// Mitsubishi GX Works2 project: ConcentricityP202112270800   PLC: Q03UDV

PROGRAM 1_AUTO
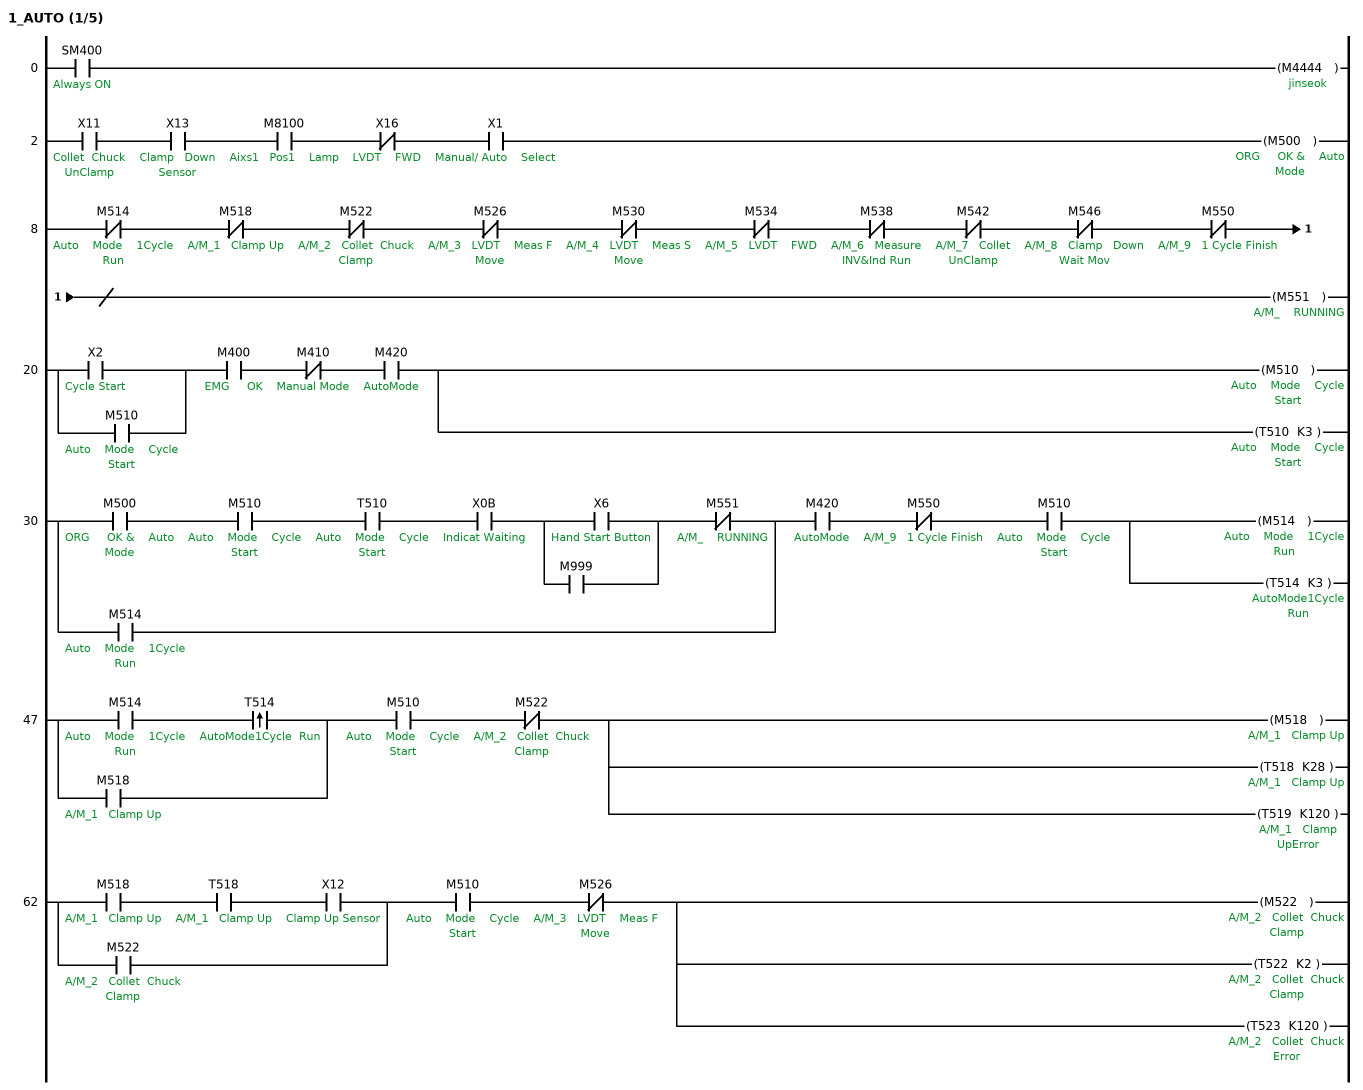
0     LD      SM400  ; Always ON
      OUT     M4444  ; jinseok
2     LD      X11  ; Collet  Chuck   UnClamp
      AND     X13  ; Clamp   Down    Sensor
      AND     M8100  ; Aixs1   Pos1    Lamp
      ANI     X16  ; LVDT    FWD
      AND     X1  ; Manual/ Auto    Select
      OUT     M500  ; ORG     OK &    Auto    Mode
8     LDI     M514  ; Auto    Mode    1Cycle  Run
      ANI     M518  ; A/M_1   Clamp Up
      ANI     M522  ; A/M_2   Collet  Chuck   Clamp
      ANI     M526  ; A/M_3   LVDT    Meas F  Move
      ANI     M530  ; A/M_4   LVDT    Meas S  Move
      ANI     M534  ; A/M_5   LVDT    FWD
      ANI     M538  ; A/M_6   Measure INV&Ind Run
      ANI     M542  ; A/M_7   Collet  UnClamp
      ANI     M546  ; A/M_8   Clamp   Down    Wait Mov
      ANI     M550  ; A/M_9   1 Cycle Finish
      INV
      OUT     M551  ; A/M_    RUNNING
20    LD      X2  ; Cycle Start
      OR      M510  ; Auto    Mode    Cycle   Start
      AND     M400  ; EMG     OK
      ANI     M410  ; Manual Mode
      AND     M420  ; AutoMode
      OUT     M510  ; Auto    Mode    Cycle   Start
      OUT     T510 K3  ; Auto    Mode    Cycle   Start
30    LD      M500  ; ORG     OK &    Auto    Mode
      AND     M510  ; Auto    Mode    Cycle   Start
      AND     T510  ; Auto    Mode    Cycle   Start
      AND     X0B  ; Indicat Waiting
      LD      X6  ; Hand Start Button
      OR      M999
      ANB
      ANI     M551  ; A/M_    RUNNING
      OR      M514  ; Auto    Mode    1Cycle  Run
      AND     M420  ; AutoMode
      ANI     M550  ; A/M_9   1 Cycle Finish
      AND     M510  ; Auto    Mode    Cycle   Start
      OUT     M514  ; Auto    Mode    1Cycle  Run
      OUT     T514 K3  ; AutoMode1Cycle  Run
47    LD      M514  ; Auto    Mode    1Cycle  Run
      ANDP    T514  ; AutoMode1Cycle  Run
      OR      M518  ; A/M_1   Clamp Up
      AND     M510  ; Auto    Mode    Cycle   Start
      ANI     M522  ; A/M_2   Collet  Chuck   Clamp
      OUT     M518  ; A/M_1   Clamp Up
      OUT     T518 K28  ; A/M_1   Clamp Up
      OUT     T519 K120  ; A/M_1   Clamp UpError
62    LD      M518  ; A/M_1   Clamp Up
      AND     T518  ; A/M_1   Clamp Up
      AND     X12  ; Clamp Up Sensor
      OR      M522  ; A/M_2   Collet  Chuck   Clamp
      AND     M510  ; Auto    Mode    Cycle   Start
      ANI     M526  ; A/M_3   LVDT    Meas F  Move
      OUT     M522  ; A/M_2   Collet  Chuck   Clamp
      OUT     T522 K2  ; A/M_2   Collet  Chuck   Clamp
      OUT     T523 K120  ; A/M_2   Collet  Chuck   Error
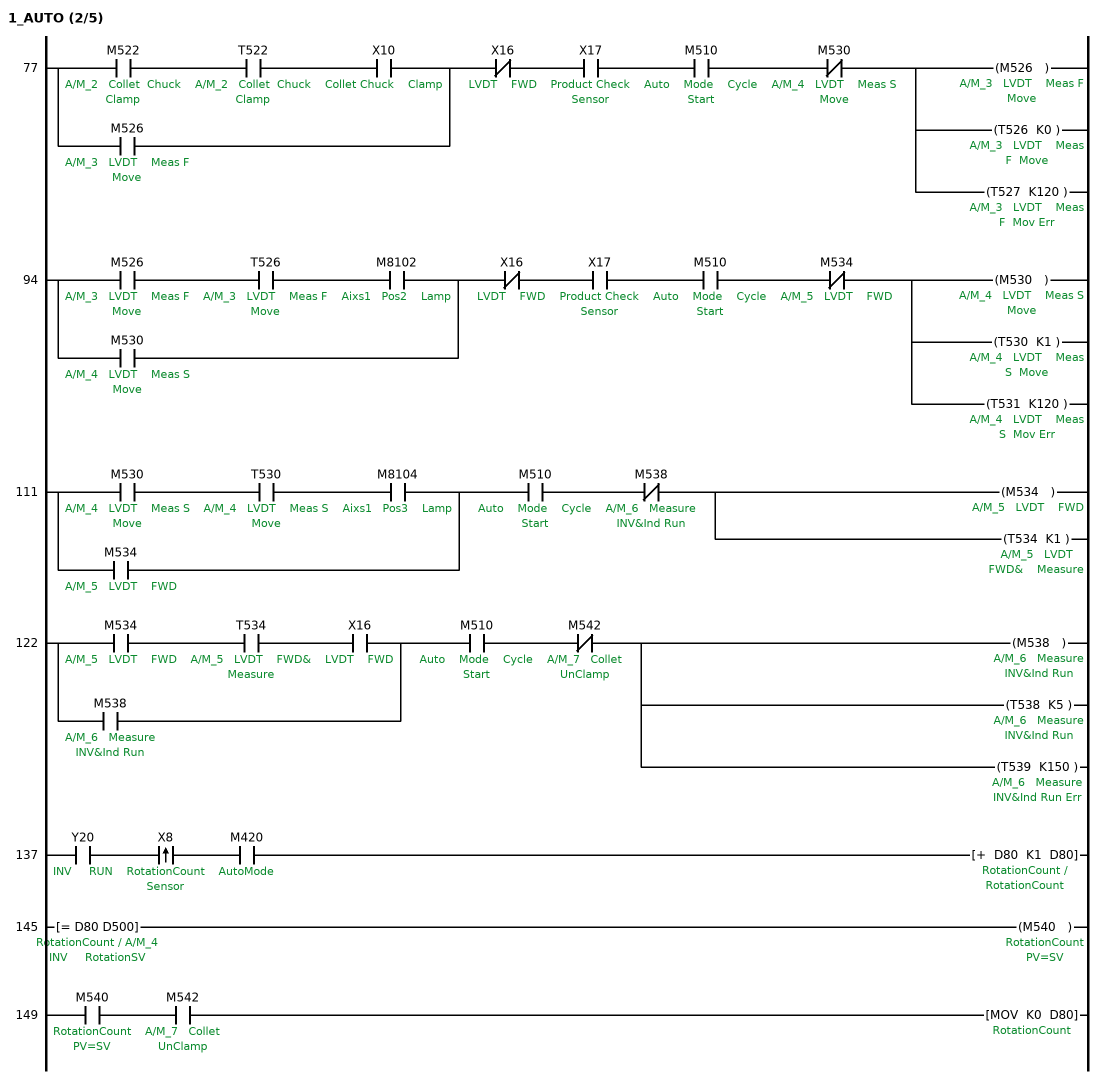
77    LD      M522  ; A/M_2   Collet  Chuck   Clamp
      AND     T522  ; A/M_2   Collet  Chuck   Clamp
      AND     X10  ; Collet Chuck    Clamp
      OR      M526  ; A/M_3   LVDT    Meas F  Move
      ANI     X16  ; LVDT    FWD
      AND     X17  ; Product Check   Sensor
      AND     M510  ; Auto    Mode    Cycle   Start
      ANI     M530  ; A/M_4   LVDT    Meas S  Move
      OUT     M526  ; A/M_3   LVDT    Meas F  Move
      OUT     T526 K0  ; A/M_3   LVDT    Meas F  Move
      OUT     T527 K120  ; A/M_3   LVDT    Meas F  Mov Err
94    LD      M526  ; A/M_3   LVDT    Meas F  Move
      AND     T526  ; A/M_3   LVDT    Meas F  Move
      AND     M8102  ; Aixs1   Pos2    Lamp
      OR      M530  ; A/M_4   LVDT    Meas S  Move
      ANI     X16  ; LVDT    FWD
      AND     X17  ; Product Check   Sensor
      AND     M510  ; Auto    Mode    Cycle   Start
      ANI     M534  ; A/M_5   LVDT    FWD
      OUT     M530  ; A/M_4   LVDT    Meas S  Move
      OUT     T530 K1  ; A/M_4   LVDT    Meas S  Move
      OUT     T531 K120  ; A/M_4   LVDT    Meas S  Mov Err
111   LD      M530  ; A/M_4   LVDT    Meas S  Move
      AND     T530  ; A/M_4   LVDT    Meas S  Move
      AND     M8104  ; Aixs1   Pos3    Lamp
      OR      M534  ; A/M_5   LVDT    FWD
      AND     M510  ; Auto    Mode    Cycle   Start
      ANI     M538  ; A/M_6   Measure INV&Ind Run
      OUT     M534  ; A/M_5   LVDT    FWD
      OUT     T534 K1  ; A/M_5   LVDT    FWD&    Measure
122   LD      M534  ; A/M_5   LVDT    FWD
      AND     T534  ; A/M_5   LVDT    FWD&    Measure
      AND     X16  ; LVDT    FWD
      OR      M538  ; A/M_6   Measure INV&Ind Run
      AND     M510  ; Auto    Mode    Cycle   Start
      ANI     M542  ; A/M_7   Collet  UnClamp
      OUT     M538  ; A/M_6   Measure INV&Ind Run
      OUT     T538 K5  ; A/M_6   Measure INV&Ind Run
      OUT     T539 K150  ; A/M_6   Measure INV&Ind Run Err
137   LD      Y20  ; INV     RUN
      ANDP    X8  ; RotationCount   Sensor
      AND     M420  ; AutoMode
      +       D80 K1 D80  ; RotationCount
145   LD=     D80 D500  ; RotationCount / A/M_4   INV     RotationSV
      OUT     M540  ; RotationCount   PV=SV
149   LD      M540  ; RotationCount   PV=SV
      AND     M542  ; A/M_7   Collet  UnClamp
      MOV     K0 D80
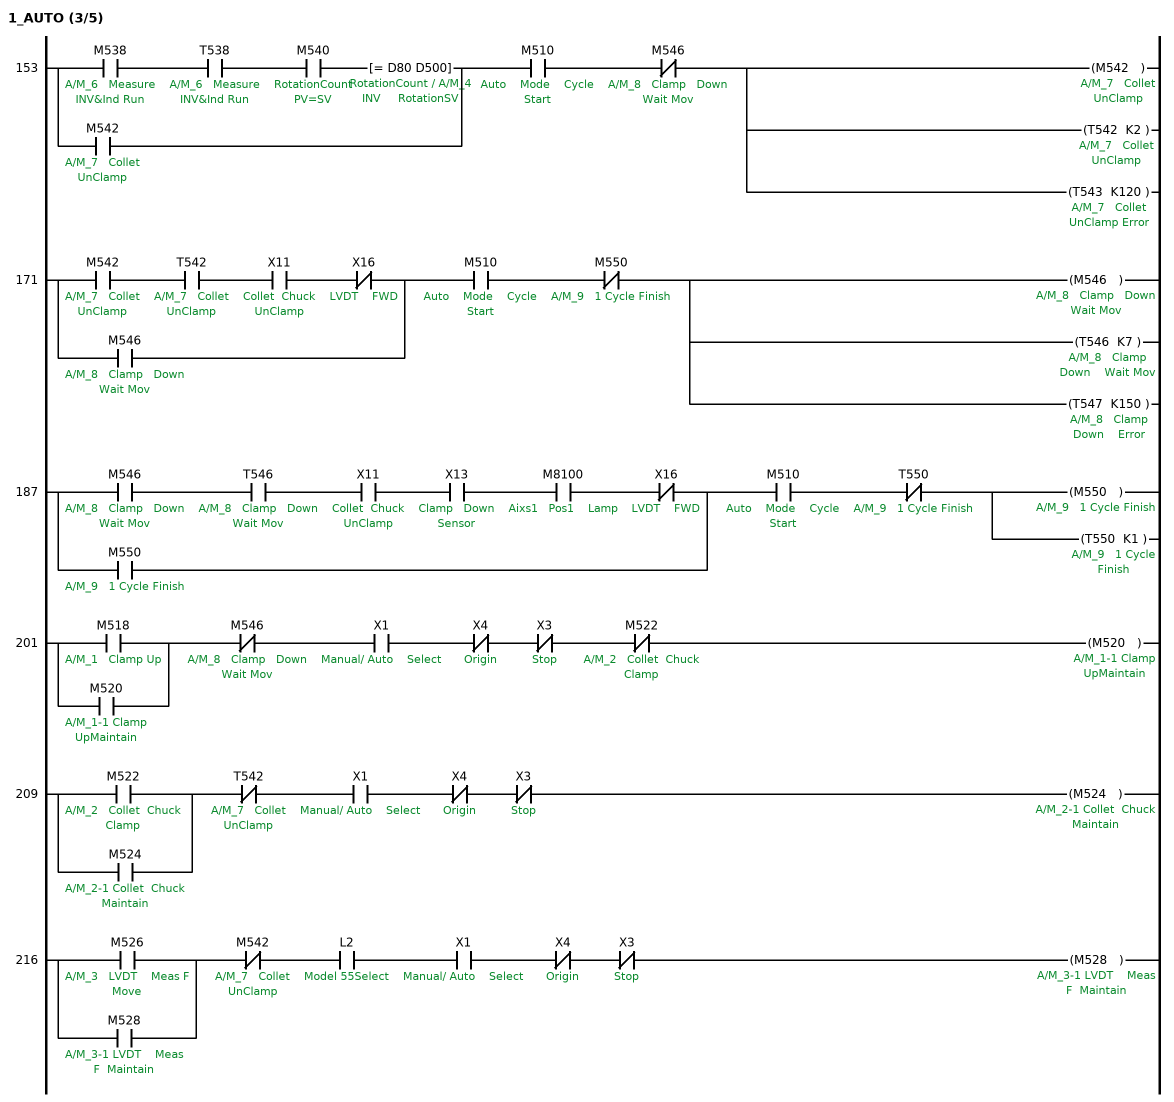
153   LD      M538  ; A/M_6   Measure INV&Ind Run
      AND     T538  ; A/M_6   Measure INV&Ind Run
      AND     M540  ; RotationCount   PV=SV
      AND=    D80 D500  ; RotationCount / A/M_4   INV     RotationSV
      OR      M542  ; A/M_7   Collet  UnClamp
      AND     M510  ; Auto    Mode    Cycle   Start
      ANI     M546  ; A/M_8   Clamp   Down    Wait Mov
      OUT     M542  ; A/M_7   Collet  UnClamp
      OUT     T542 K2  ; A/M_7   Collet  UnClamp
      OUT     T543 K120  ; A/M_7   Collet  UnClamp Error
171   LD      M542  ; A/M_7   Collet  UnClamp
      AND     T542  ; A/M_7   Collet  UnClamp
      AND     X11  ; Collet  Chuck   UnClamp
      ANI     X16  ; LVDT    FWD
      OR      M546  ; A/M_8   Clamp   Down    Wait Mov
      AND     M510  ; Auto    Mode    Cycle   Start
      ANI     M550  ; A/M_9   1 Cycle Finish
      OUT     M546  ; A/M_8   Clamp   Down    Wait Mov
      OUT     T546 K7  ; A/M_8   Clamp   Down    Wait Mov
      OUT     T547 K150  ; A/M_8   Clamp   Down    Error
187   LD      M546  ; A/M_8   Clamp   Down    Wait Mov
      AND     T546  ; A/M_8   Clamp   Down    Wait Mov
      AND     X11  ; Collet  Chuck   UnClamp
      AND     X13  ; Clamp   Down    Sensor
      AND     M8100  ; Aixs1   Pos1    Lamp
      ANI     X16  ; LVDT    FWD
      OR      M550  ; A/M_9   1 Cycle Finish
      AND     M510  ; Auto    Mode    Cycle   Start
      ANI     T550  ; A/M_9   1 Cycle Finish
      OUT     M550  ; A/M_9   1 Cycle Finish
      OUT     T550 K1  ; A/M_9   1 Cycle Finish
201   LD      M518  ; A/M_1   Clamp Up
      OR      M520  ; A/M_1-1 Clamp UpMaintain
      ANI     M546  ; A/M_8   Clamp   Down    Wait Mov
      AND     X1  ; Manual/ Auto    Select
      ANI     X4  ; Origin
      ANI     X3  ; Stop
      ANI     M522  ; A/M_2   Collet  Chuck   Clamp
      OUT     M520  ; A/M_1-1 Clamp UpMaintain
209   LD      M522  ; A/M_2   Collet  Chuck   Clamp
      OR      M524  ; A/M_2-1 Collet  Chuck   Maintain
      ANI     T542  ; A/M_7   Collet  UnClamp
      AND     X1  ; Manual/ Auto    Select
      ANI     X4  ; Origin
      ANI     X3  ; Stop
      OUT     M524  ; A/M_2-1 Collet  Chuck   Maintain
216   LD      M526  ; A/M_3   LVDT    Meas F  Move
      OR      M528  ; A/M_3-1 LVDT    Meas F  Maintain
      ANI     M542  ; A/M_7   Collet  UnClamp
      AND     L2  ; Model 55Select
      AND     X1  ; Manual/ Auto    Select
      ANI     X4  ; Origin
      ANI     X3  ; Stop
      OUT     M528  ; A/M_3-1 LVDT    Meas F  Maintain
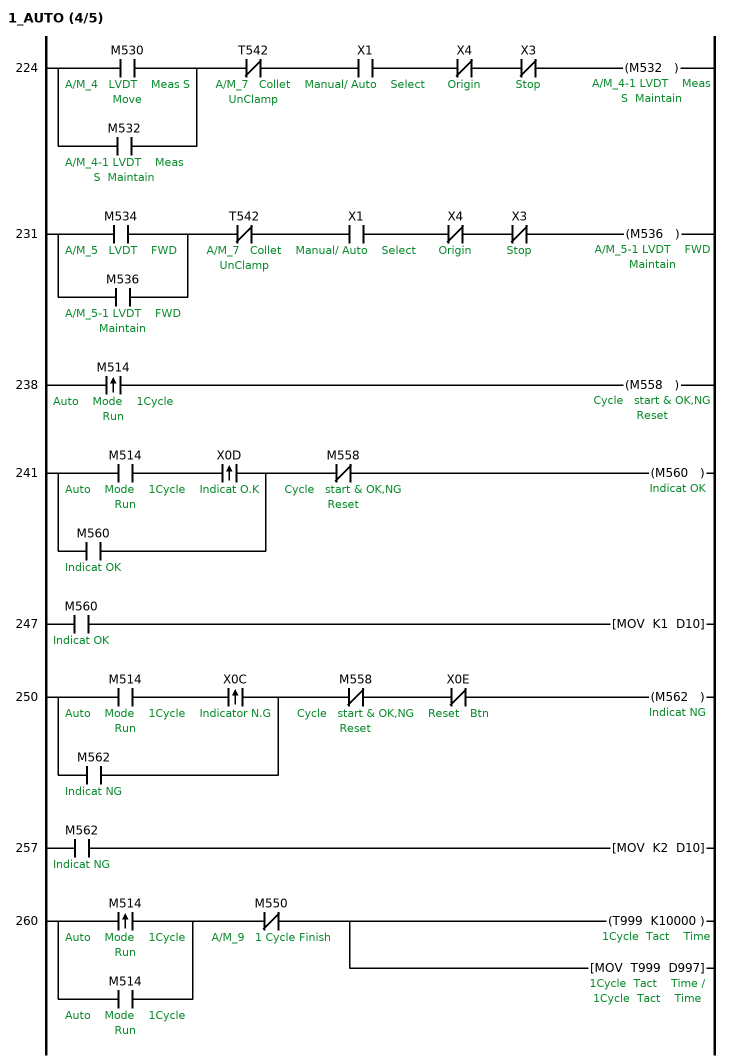
224   LD      M530  ; A/M_4   LVDT    Meas S  Move
      OR      M532  ; A/M_4-1 LVDT    Meas S  Maintain
      ANI     T542  ; A/M_7   Collet  UnClamp
      AND     X1  ; Manual/ Auto    Select
      ANI     X4  ; Origin
      ANI     X3  ; Stop
      OUT     M532  ; A/M_4-1 LVDT    Meas S  Maintain
231   LD      M534  ; A/M_5   LVDT    FWD
      OR      M536  ; A/M_5-1 LVDT    FWD     Maintain
      ANI     T542  ; A/M_7   Collet  UnClamp
      AND     X1  ; Manual/ Auto    Select
      ANI     X4  ; Origin
      ANI     X3  ; Stop
      OUT     M536  ; A/M_5-1 LVDT    FWD     Maintain
238   LDP     M514  ; Auto    Mode    1Cycle  Run
      OUT     M558  ; Cycle   start & OK,NG   Reset
241   LD      M514  ; Auto    Mode    1Cycle  Run
      ANDP    X0D  ; Indicat O.K
      OR      M560  ; Indicat OK
      ANI     M558  ; Cycle   start & OK,NG   Reset
      OUT     M560  ; Indicat OK
247   LD      M560  ; Indicat OK
      MOV     K1 D10
250   LD      M514  ; Auto    Mode    1Cycle  Run
      ANDP    X0C  ; Indicator N.G
      OR      M562  ; Indicat NG
      ANI     M558  ; Cycle   start & OK,NG   Reset
      ANI     X0E  ; Reset   Btn
      OUT     M562  ; Indicat NG
257   LD      M562  ; Indicat NG
      MOV     K2 D10
260   LDP     M514  ; Auto    Mode    1Cycle  Run
      OR      M514  ; Auto    Mode    1Cycle  Run
      ANI     M550  ; A/M_9   1 Cycle Finish
      OUT     T999 K10000  ; 1Cycle  Tact    Time
      MOV     T999 D997  ; 1Cycle  Tact    Time
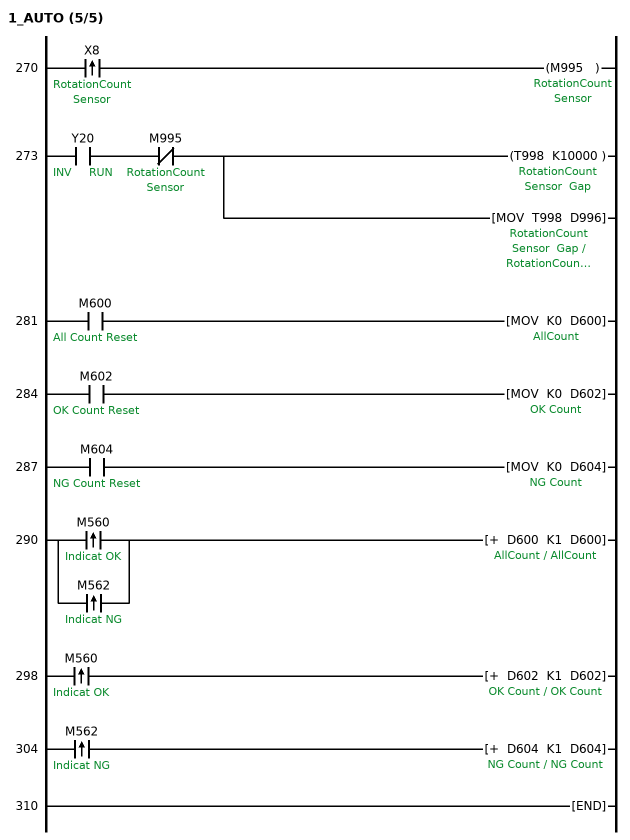
270   LDP     X8  ; RotationCount   Sensor
      OUT     M995  ; RotationCount   Sensor
273   LD      Y20  ; INV     RUN
      ANI     M995  ; RotationCount   Sensor
      OUT     T998 K10000  ; RotationCount   Sensor  Gap
      MOV     T998 D996  ; RotationCount   Sensor  Gap
281   LD      M600  ; All Count Reset
      MOV     K0 D600  ; AllCount
284   LD      M602  ; OK Count Reset
      MOV     K0 D602  ; OK Count
287   LD      M604  ; NG Count Reset
      MOV     K0 D604  ; NG Count
290   LDP     M560  ; Indicat OK
      ORP     M562  ; Indicat NG
      +       D600 K1 D600
298   LDP     M560  ; Indicat OK
      +       D602 K1 D602
304   LDP     M562  ; Indicat NG
      +       D604 K1 D604
310   END
END_PROGRAM

PROGRAM 2_MANUAL
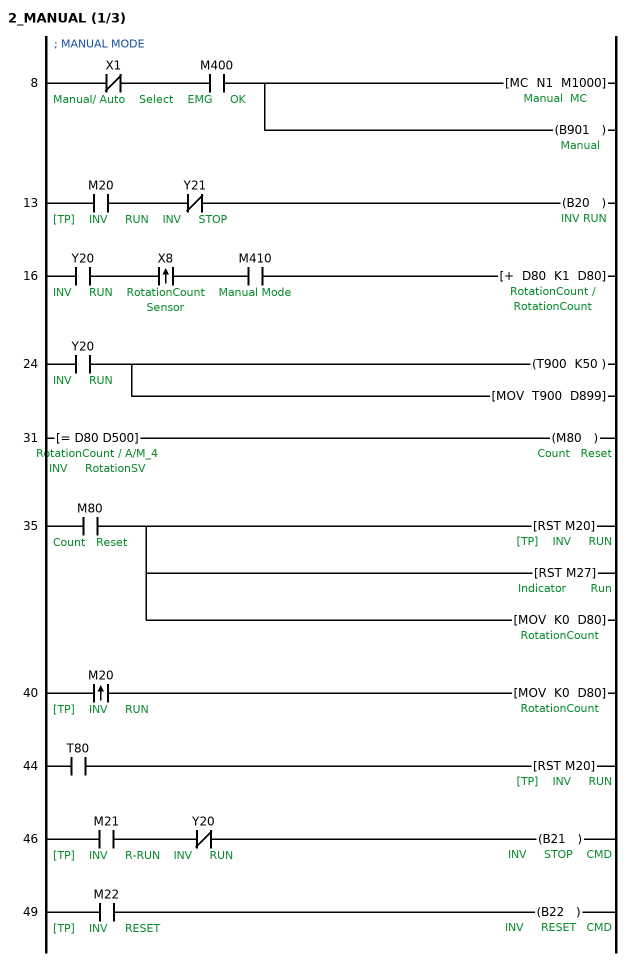
; MANUAL MODE
8     LDI     X1  ; Manual/ Auto    Select
      AND     M400  ; EMG     OK
      MC      N1 M1000  ; Manual  MC
      OUT     B901  ; Manual
13    LD      M20  ; [TP]    INV     RUN
      ANI     Y21  ; INV     STOP
      OUT     B20  ; INV RUN
16    LD      Y20  ; INV     RUN
      ANDP    X8  ; RotationCount   Sensor
      AND     M410  ; Manual Mode
      +       D80 K1 D80  ; RotationCount
24    LD      Y20  ; INV     RUN
      OUT     T900 K50
      MOV     T900 D899
31    LD=     D80 D500  ; RotationCount / A/M_4   INV     RotationSV
      OUT     M80  ; Count   Reset
35    LD      M80  ; Count   Reset
      RST     M20  ; [TP]    INV     RUN
      RST     M27  ; Indicator       Run
      MOV     K0 D80
40    LDP     M20  ; [TP]    INV     RUN
      MOV     K0 D80
44    LD      T80
      RST     M20  ; [TP]    INV     RUN
46    LD      M21  ; [TP]    INV     R-RUN
      ANI     Y20  ; INV     RUN
      OUT     B21  ; INV     STOP    CMD
49    LD      M22  ; [TP]    INV     RESET
      OUT     B22  ; INV     RESET   CMD
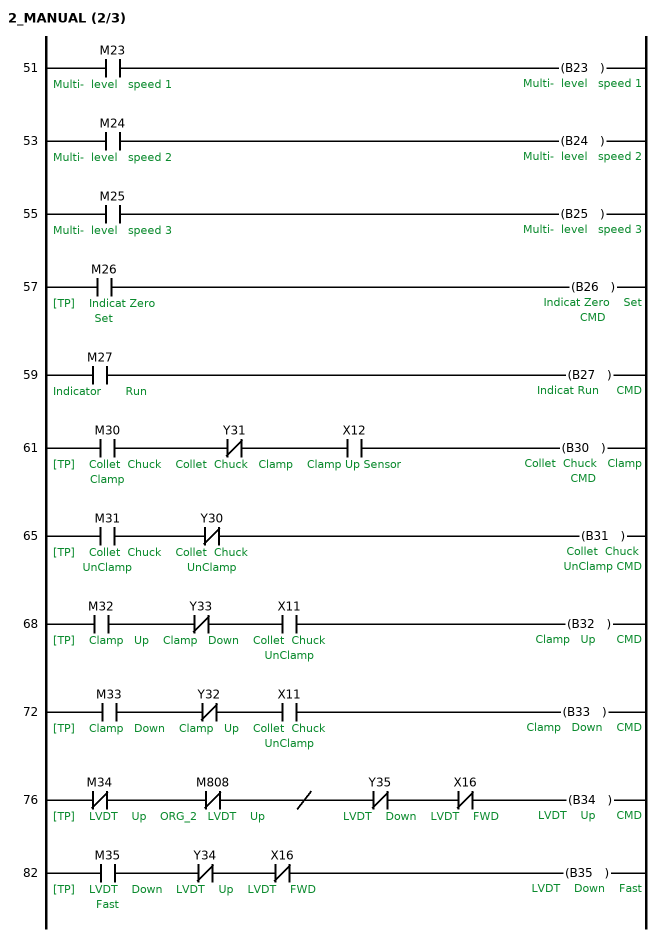
51    LD      M23  ; Multi-  level   speed 1
      OUT     B23  ; Multi-  level   speed 1
53    LD      M24  ; Multi-  level   speed 2
      OUT     B24  ; Multi-  level   speed 2
55    LD      M25  ; Multi-  level   speed 3
      OUT     B25  ; Multi-  level   speed 3
57    LD      M26  ; [TP]    Indicat Zero    Set
      OUT     B26  ; Indicat Zero    Set     CMD
59    LD      M27  ; Indicator       Run
      OUT     B27  ; Indicat Run     CMD
61    LD      M30  ; [TP]    Collet  Chuck   Clamp
      ANI     Y31  ; Collet  Chuck   Clamp
      AND     X12  ; Clamp Up Sensor
      OUT     B30  ; Collet  Chuck   Clamp   CMD
65    LD      M31  ; [TP]    Collet  Chuck   UnClamp
      ANI     Y30  ; Collet  Chuck   UnClamp
      OUT     B31  ; Collet  Chuck   UnClamp CMD
68    LD      M32  ; [TP]    Clamp   Up
      ANI     Y33  ; Clamp   Down
      AND     X11  ; Collet  Chuck   UnClamp
      OUT     B32  ; Clamp   Up      CMD
72    LD      M33  ; [TP]    Clamp   Down
      ANI     Y32  ; Clamp   Up
      AND     X11  ; Collet  Chuck   UnClamp
      OUT     B33  ; Clamp   Down    CMD
76    LDI     M34  ; [TP]    LVDT    Up
      ANI     M808  ; ORG_2   LVDT    Up
      INV
      ANI     Y35  ; LVDT    Down
      ANI     X16  ; LVDT    FWD
      OUT     B34  ; LVDT    Up      CMD
82    LD      M35  ; [TP]    LVDT    Down    Fast
      ANI     Y34  ; LVDT    Up
      ANI     X16  ; LVDT    FWD
      OUT     B35  ; LVDT    Down    Fast
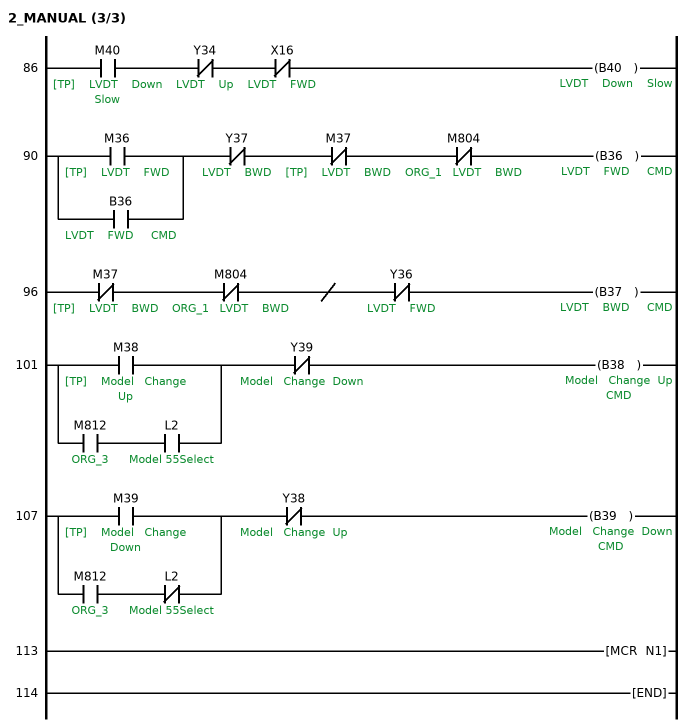
86    LD      M40  ; [TP]    LVDT    Down    Slow
      ANI     Y34  ; LVDT    Up
      ANI     X16  ; LVDT    FWD
      OUT     B40  ; LVDT    Down    Slow
90    LD      M36  ; [TP]    LVDT    FWD
      OR      B36  ; LVDT    FWD     CMD
      ANI     Y37  ; LVDT    BWD
      ANI     M37  ; [TP]    LVDT    BWD
      ANI     M804  ; ORG_1   LVDT    BWD
      OUT     B36  ; LVDT    FWD     CMD
96    LDI     M37  ; [TP]    LVDT    BWD
      ANI     M804  ; ORG_1   LVDT    BWD
      INV
      ANI     Y36  ; LVDT    FWD
      OUT     B37  ; LVDT    BWD     CMD
101   LD      M38  ; [TP]    Model   Change  Up
      LD      M812  ; ORG_3
      AND     L2  ; Model 55Select
      ORB
      ANI     Y39  ; Model   Change  Down
      OUT     B38  ; Model   Change  Up      CMD
107   LD      M39  ; [TP]    Model   Change  Down
      LD      M812  ; ORG_3
      ANI     L2  ; Model 55Select
      ORB
      ANI     Y38  ; Model   Change  Up
      OUT     B39  ; Model   Change  Down    CMD
113   MCR     N1
114   END
END_PROGRAM

PROGRAM 700_LVDT
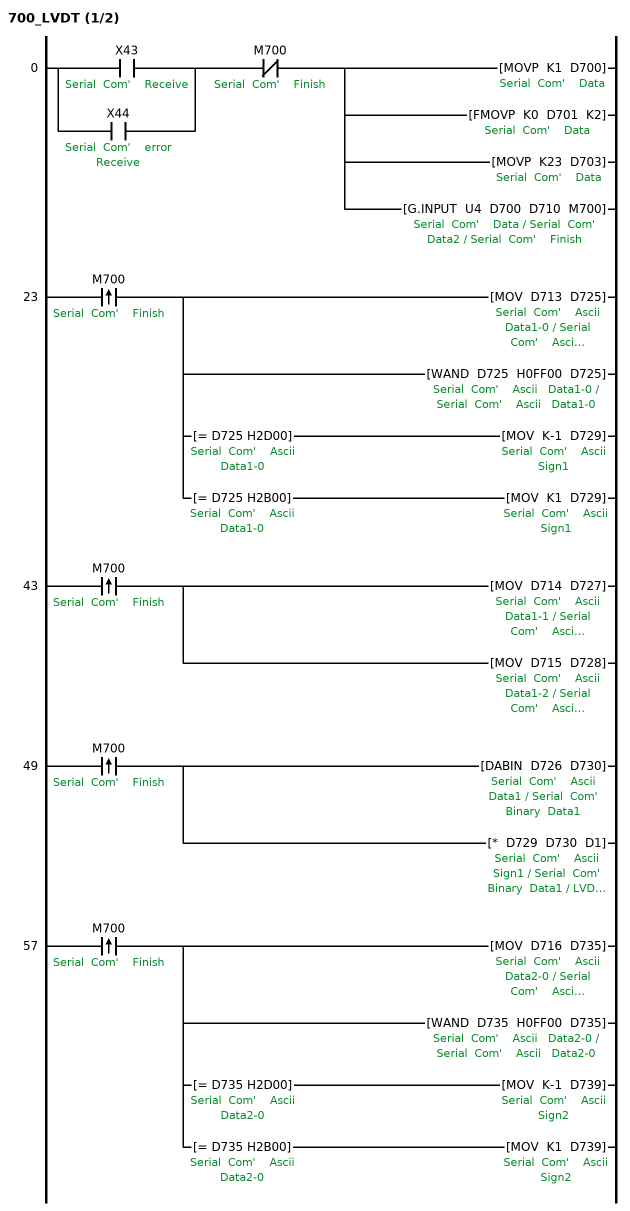
0     LD      X43  ; Serial  Com'    Receive
      OR      X44  ; Serial  Com'    error   Receive
      ANI     M700  ; Serial  Com'    Finish
      MOVP    K1 D700  ; Serial  Com'    Data
      FMOVP   K0 D701 K2  ; Serial  Com'    Data
      MOVP    K23 D703  ; Serial  Com'    Data
      G.INPUT U4 D700 D710 M700  ; Serial  Com'    Data2
23    LDP     M700  ; Serial  Com'    Finish
      MOV     D713 D725  ; Serial  Com'    Ascii   Data1-0 / Serial  Com'    Ascii   Data1-0
      WAND    D725 H0FF00 D725
      MPS
      AND=    D725 H2D00  ; Serial  Com'    Ascii   Data1-0
      MOV     K-1 D729  ; Serial  Com'    Ascii   Sign1
      MPP
      AND=    D725 H2B00  ; Serial  Com'    Ascii   Data1-0
      MOV     K1 D729
43    LDP     M700  ; Serial  Com'    Finish
      MOV     D714 D727  ; Serial  Com'    Ascii   Data1-1 / Serial  Com'    Ascii   Data1-1
      MOV     D715 D728  ; Serial  Com'    Ascii   Data1-2 / Serial  Com'    Ascii   Data1-2
49    LDP     M700  ; Serial  Com'    Finish
      DABIN   D726 D730  ; Serial  Com'    Ascii   Data1 / Serial  Com'    Binary  Data1
      *       D729 D730 D1  ; LVDT 1stDATA
57    LDP     M700  ; Serial  Com'    Finish
      MOV     D716 D735  ; Serial  Com'    Ascii   Data2-0 / Serial  Com'    Ascii   Data2-0
      WAND    D735 H0FF00 D735
      MPS
      AND=    D735 H2D00  ; Serial  Com'    Ascii   Data2-0
      MOV     K-1 D739  ; Serial  Com'    Ascii   Sign2
      MPP
      AND=    D735 H2B00  ; Serial  Com'    Ascii   Data2-0
      MOV     K1 D739
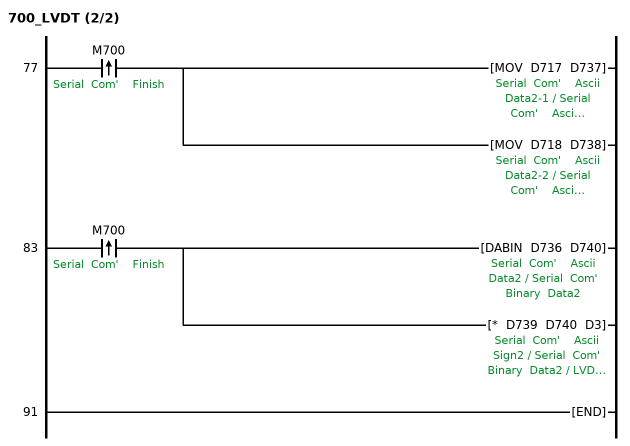
77    LDP     M700  ; Serial  Com'    Finish
      MOV     D717 D737  ; Serial  Com'    Ascii   Data2-1 / Serial  Com'    Ascii   Data2-1
      MOV     D718 D738  ; Serial  Com'    Ascii   Data2-2 / Serial  Com'    Ascii   Data2-2
83    LDP     M700  ; Serial  Com'    Finish
      DABIN   D736 D740  ; Serial  Com'    Ascii   Data2 / Serial  Com'    Binary  Data2
      *       D739 D740 D3  ; LVDT 2ndDATA
91    END
END_PROGRAM

PROGRAM 5_ALARM
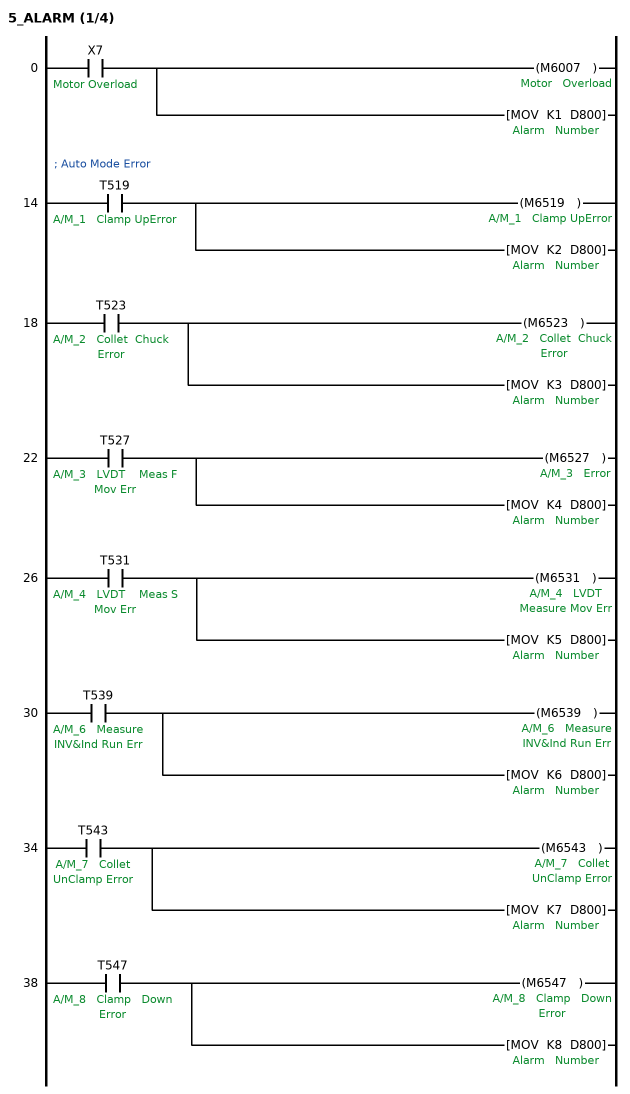
0     LD      X7  ; Motor Overload
      OUT     M6007  ; Motor   Overload
      MOV     K1 D800  ; Alarm   Number
; Auto Mode Error
14    LD      T519  ; A/M_1   Clamp UpError
      OUT     M6519  ; A/M_1   Clamp UpError
      MOV     K2 D800
18    LD      T523  ; A/M_2   Collet  Chuck   Error
      OUT     M6523  ; A/M_2   Collet  Chuck   Error
      MOV     K3 D800
22    LD      T527  ; A/M_3   LVDT    Meas F  Mov Err
      OUT     M6527  ; A/M_3   Error
      MOV     K4 D800
26    LD      T531  ; A/M_4   LVDT    Meas S  Mov Err
      OUT     M6531  ; A/M_4   LVDT    Measure Mov Err
      MOV     K5 D800
30    LD      T539  ; A/M_6   Measure INV&Ind Run Err
      OUT     M6539  ; A/M_6   Measure INV&Ind Run Err
      MOV     K6 D800
34    LD      T543  ; A/M_7   Collet  UnClamp Error
      OUT     M6543  ; A/M_7   Collet  UnClamp Error
      MOV     K7 D800
38    LD      T547  ; A/M_8   Clamp   Down    Error
      OUT     M6547  ; A/M_8   Clamp   Down    Error
      MOV     K8 D800
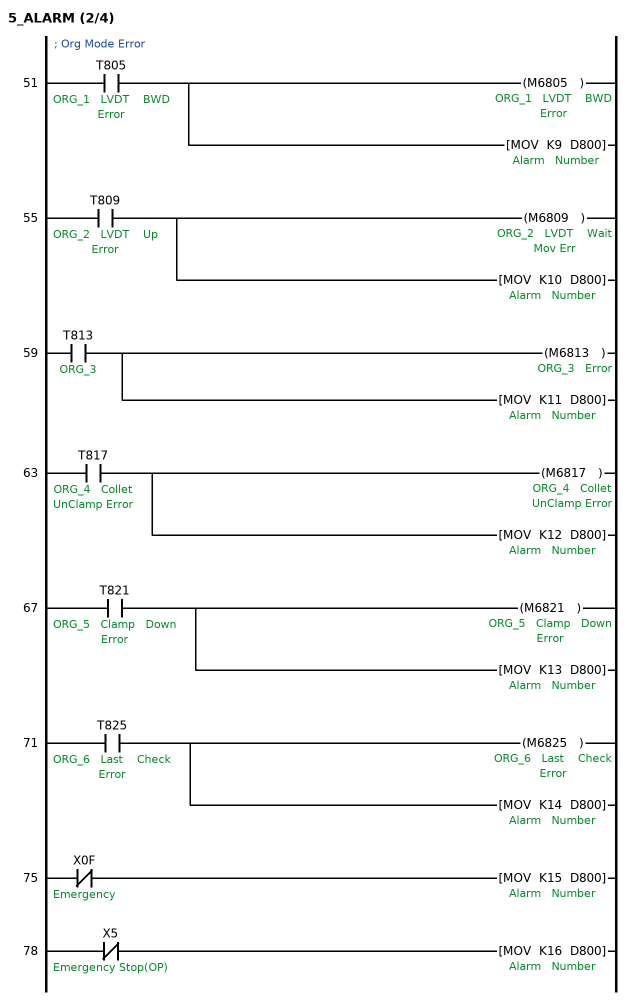
; Org Mode Error
51    LD      T805  ; ORG_1   LVDT    BWD     Error
      OUT     M6805  ; ORG_1   LVDT    BWD     Error
      MOV     K9 D800
55    LD      T809  ; ORG_2   LVDT    Up      Error
      OUT     M6809  ; ORG_2   LVDT    Wait    Mov Err
      MOV     K10 D800
59    LD      T813  ; ORG_3
      OUT     M6813  ; ORG_3   Error
      MOV     K11 D800
63    LD      T817  ; ORG_4   Collet  UnClamp Error
      OUT     M6817  ; ORG_4   Collet  UnClamp Error
      MOV     K12 D800
67    LD      T821  ; ORG_5   Clamp   Down    Error
      OUT     M6821  ; ORG_5   Clamp   Down    Error
      MOV     K13 D800
71    LD      T825  ; ORG_6   Last    Check   Error
      OUT     M6825  ; ORG_6   Last    Check   Error
      MOV     K14 D800
75    LDI     X0F  ; Emergency
      MOV     K15 D800
78    LDI     X5  ; Emergency Stop(OP)
      MOV     K16 D800
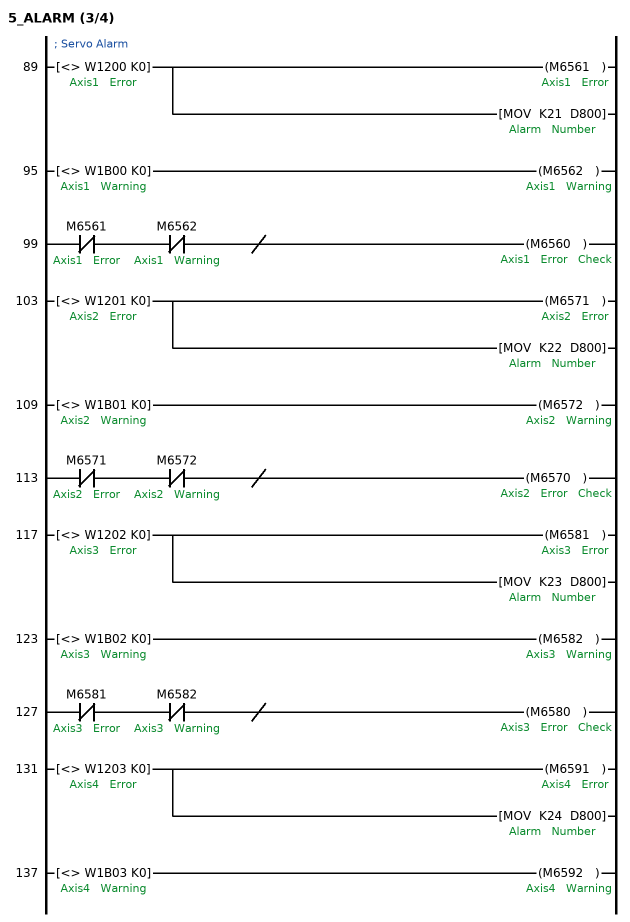
; Servo Alarm
89    LD<>    W1200 K0  ; Axis1   Error
      OUT     M6561  ; Axis1   Error
      MOV     K21 D800
95    LD<>    W1B00 K0  ; Axis1   Warning
      OUT     M6562  ; Axis1   Warning
99    LDI     M6561  ; Axis1   Error
      ANI     M6562  ; Axis1   Warning
      INV
      OUT     M6560  ; Axis1   Error   Check
103   LD<>    W1201 K0  ; Axis2   Error
      OUT     M6571  ; Axis2   Error
      MOV     K22 D800
109   LD<>    W1B01 K0  ; Axis2   Warning
      OUT     M6572  ; Axis2   Warning
113   LDI     M6571  ; Axis2   Error
      ANI     M6572  ; Axis2   Warning
      INV
      OUT     M6570  ; Axis2   Error   Check
117   LD<>    W1202 K0  ; Axis3   Error
      OUT     M6581  ; Axis3   Error
      MOV     K23 D800
123   LD<>    W1B02 K0  ; Axis3   Warning
      OUT     M6582  ; Axis3   Warning
127   LDI     M6581  ; Axis3   Error
      ANI     M6582  ; Axis3   Warning
      INV
      OUT     M6580  ; Axis3   Error   Check
131   LD<>    W1203 K0  ; Axis4   Error
      OUT     M6591  ; Axis4   Error
      MOV     K24 D800
137   LD<>    W1B03 K0  ; Axis4   Warning
      OUT     M6592  ; Axis4   Warning
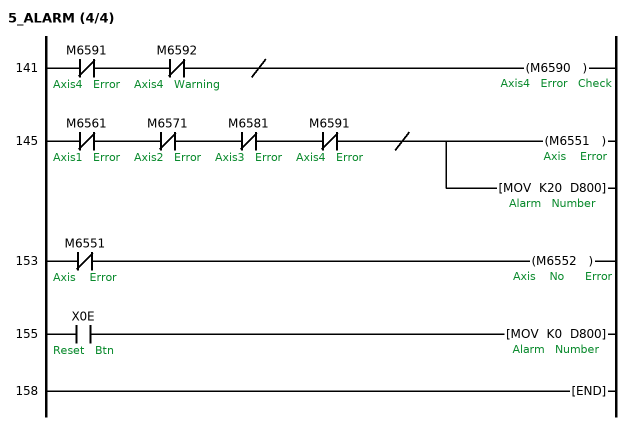
141   LDI     M6591  ; Axis4   Error
      ANI     M6592  ; Axis4   Warning
      INV
      OUT     M6590  ; Axis4   Error   Check
145   LDI     M6561  ; Axis1   Error
      ANI     M6571  ; Axis2   Error
      ANI     M6581  ; Axis3   Error
      ANI     M6591  ; Axis4   Error
      INV
      OUT     M6551  ; Axis    Error
      MOV     K20 D800
153   LDI     M6551  ; Axis    Error
      OUT     M6552  ; Axis    No      Error
155   LD      X0E  ; Reset   Btn
      MOV     K0 D800
158   END
END_PROGRAM

PROGRAM 6_OUTPUT
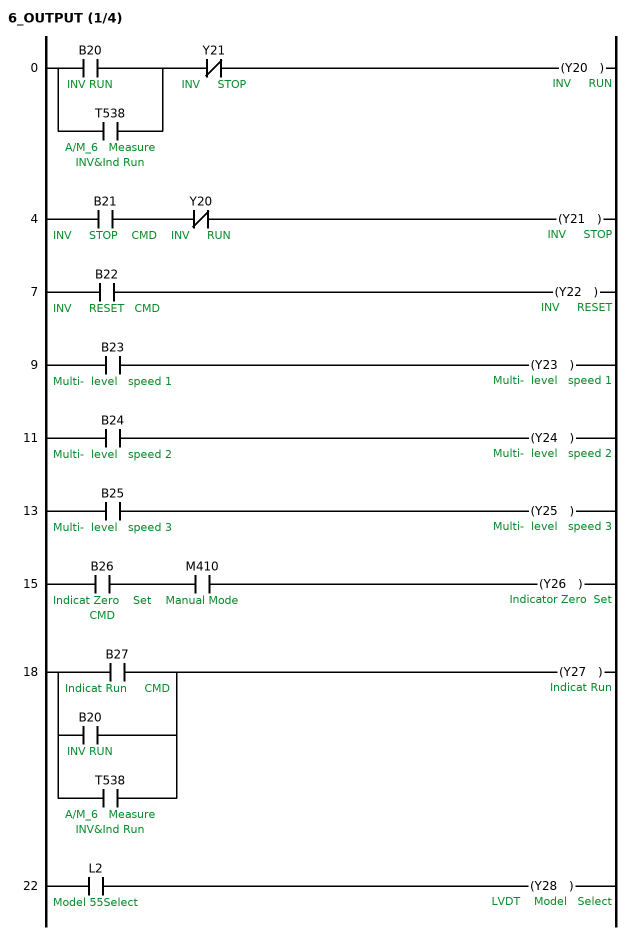
0     LD      B20  ; INV RUN
      OR      T538  ; A/M_6   Measure INV&Ind Run
      ANI     Y21  ; INV     STOP
      OUT     Y20  ; INV     RUN
4     LD      B21  ; INV     STOP    CMD
      ANI     Y20  ; INV     RUN
      OUT     Y21  ; INV     STOP
7     LD      B22  ; INV     RESET   CMD
      OUT     Y22  ; INV     RESET
9     LD      B23  ; Multi-  level   speed 1
      OUT     Y23  ; Multi-  level   speed 1
11    LD      B24  ; Multi-  level   speed 2
      OUT     Y24  ; Multi-  level   speed 2
13    LD      B25  ; Multi-  level   speed 3
      OUT     Y25  ; Multi-  level   speed 3
15    LD      B26  ; Indicat Zero    Set     CMD
      AND     M410  ; Manual Mode
      OUT     Y26  ; Indicator Zero  Set
18    LD      B27  ; Indicat Run     CMD
      OR      B20  ; INV RUN
      OR      T538  ; A/M_6   Measure INV&Ind Run
      OUT     Y27  ; Indicat Run
22    LD      L2  ; Model 55Select
      OUT     Y28  ; LVDT    Model   Select
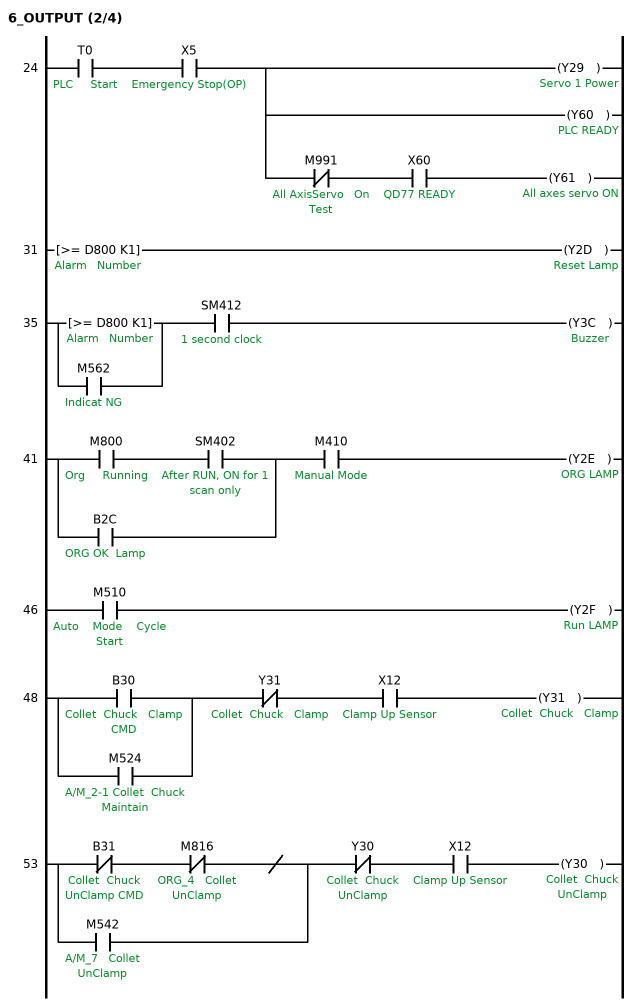
24    LD      T0  ; PLC     Start
      AND     X5  ; Emergency Stop(OP)
      OUT     Y29  ; Servo 1 Power
      OUT     Y60  ; PLC READY
      ANI     M991  ; All AxisServo   On      Test
      AND     X60  ; QD77 READY
      OUT     Y61  ; All axes servo ON
31    LD>=    D800 K1  ; Alarm   Number
      OUT     Y2D  ; Reset Lamp
35    LD>=    D800 K1  ; Alarm   Number
      OR      M562  ; Indicat NG
      AND     SM412  ; 1 second clock
      OUT     Y3C  ; Buzzer
41    LD      M800  ; Org     Running
      AND     SM402  ; After RUN, ON for 1 scan only
      OR      B2C  ; ORG OK  Lamp
      AND     M410  ; Manual Mode
      OUT     Y2E  ; ORG LAMP
46    LD      M510  ; Auto    Mode    Cycle   Start
      OUT     Y2F  ; Run LAMP
48    LD      B30  ; Collet  Chuck   Clamp   CMD
      OR      M524  ; A/M_2-1 Collet  Chuck   Maintain
      ANI     Y31  ; Collet  Chuck   Clamp
      AND     X12  ; Clamp Up Sensor
      OUT     Y31  ; Collet  Chuck   Clamp
53    LDI     B31  ; Collet  Chuck   UnClamp CMD
      ANI     M816  ; ORG_4   Collet  UnClamp
      INV
      OR      M542  ; A/M_7   Collet  UnClamp
      ANI     Y30  ; Collet  Chuck   UnClamp
      AND     X12  ; Clamp Up Sensor
      OUT     Y30  ; Collet  Chuck   UnClamp
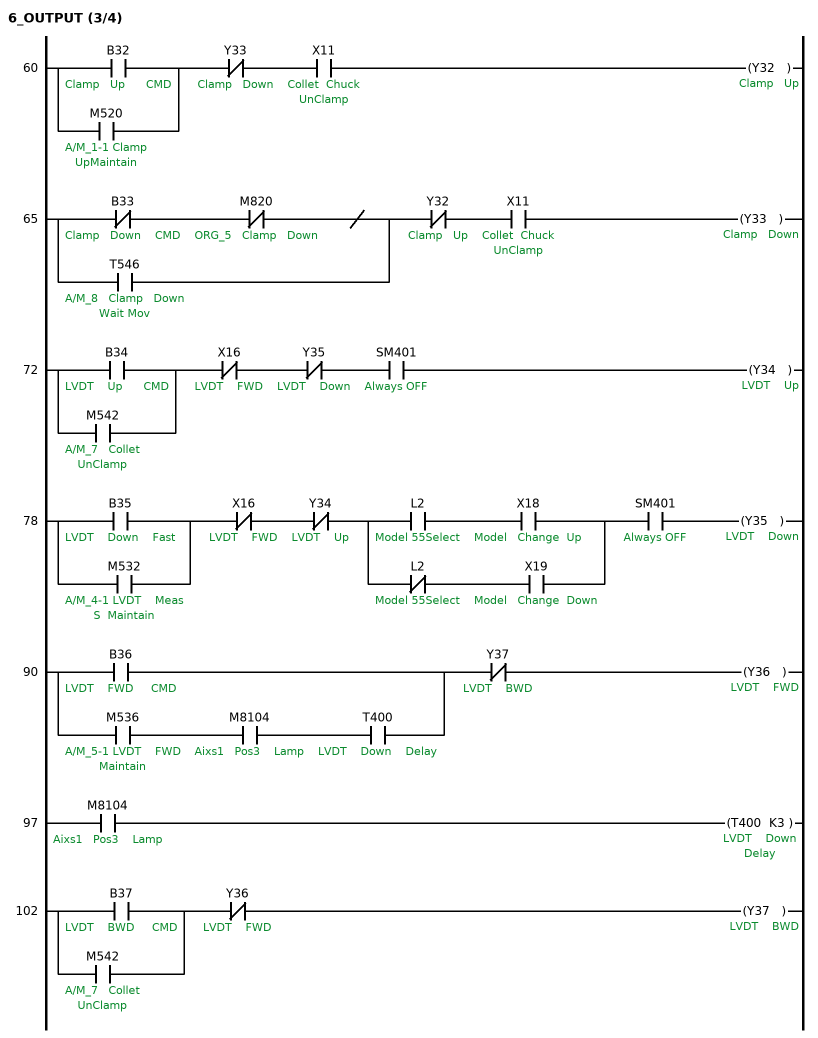
60    LD      B32  ; Clamp   Up      CMD
      OR      M520  ; A/M_1-1 Clamp UpMaintain
      ANI     Y33  ; Clamp   Down
      AND     X11  ; Collet  Chuck   UnClamp
      OUT     Y32  ; Clamp   Up
65    LDI     B33  ; Clamp   Down    CMD
      ANI     M820  ; ORG_5   Clamp   Down
      INV
      OR      T546  ; A/M_8   Clamp   Down    Wait Mov
      ANI     Y32  ; Clamp   Up
      AND     X11  ; Collet  Chuck   UnClamp
      OUT     Y33  ; Clamp   Down
72    LD      B34  ; LVDT    Up      CMD
      OR      M542  ; A/M_7   Collet  UnClamp
      ANI     X16  ; LVDT    FWD
      ANI     Y35  ; LVDT    Down
      AND     SM401  ; Always OFF
      OUT     Y34  ; LVDT    Up
78    LD      B35  ; LVDT    Down    Fast
      OR      M532  ; A/M_4-1 LVDT    Meas S  Maintain
      ANI     X16  ; LVDT    FWD
      ANI     Y34  ; LVDT    Up
      LD      L2  ; Model 55Select
      AND     X18  ; Model   Change  Up
      LDI     L2  ; Model 55Select
      AND     X19  ; Model   Change  Down
      ORB
      ANB
      AND     SM401  ; Always OFF
      OUT     Y35  ; LVDT    Down
90    LD      B36  ; LVDT    FWD     CMD
      LD      M536  ; A/M_5-1 LVDT    FWD     Maintain
      AND     M8104  ; Aixs1   Pos3    Lamp
      AND     T400  ; LVDT    Down    Delay
      ORB
      ANI     Y37  ; LVDT    BWD
      OUT     Y36  ; LVDT    FWD
97    LD      M8104  ; Aixs1   Pos3    Lamp
      OUT     T400 K3  ; LVDT    Down    Delay
102   LD      B37  ; LVDT    BWD     CMD
      OR      M542  ; A/M_7   Collet  UnClamp
      ANI     Y36  ; LVDT    FWD
      OUT     Y37  ; LVDT    BWD
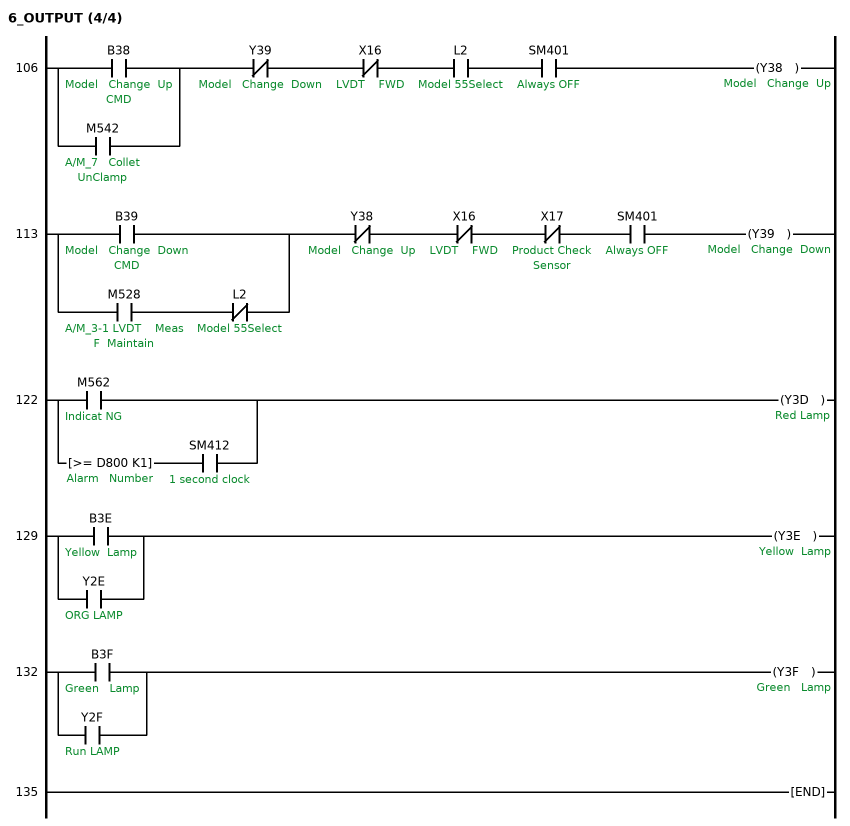
106   LD      B38  ; Model   Change  Up      CMD
      OR      M542  ; A/M_7   Collet  UnClamp
      ANI     Y39  ; Model   Change  Down
      ANI     X16  ; LVDT    FWD
      AND     L2  ; Model 55Select
      AND     SM401  ; Always OFF
      OUT     Y38  ; Model   Change  Up
113   LD      B39  ; Model   Change  Down    CMD
      LD      M528  ; A/M_3-1 LVDT    Meas F  Maintain
      ANI     L2  ; Model 55Select
      ORB
      ANI     Y38  ; Model   Change  Up
      ANI     X16  ; LVDT    FWD
      ANI     X17  ; Product Check   Sensor
      AND     SM401  ; Always OFF
      OUT     Y39  ; Model   Change  Down
122   LD      M562  ; Indicat NG
      LD>=    D800 K1  ; Alarm   Number
      AND     SM412  ; 1 second clock
      ORB
      OUT     Y3D  ; Red Lamp
129   LD      B3E  ; Yellow  Lamp
      OR      Y2E  ; ORG LAMP
      OUT     Y3E  ; Yellow  Lamp
132   LD      B3F  ; Green   Lamp
      OR      Y2F  ; Run LAMP
      OUT     Y3F  ; Green   Lamp
135   END
END_PROGRAM

PROGRAM 0_MAIN
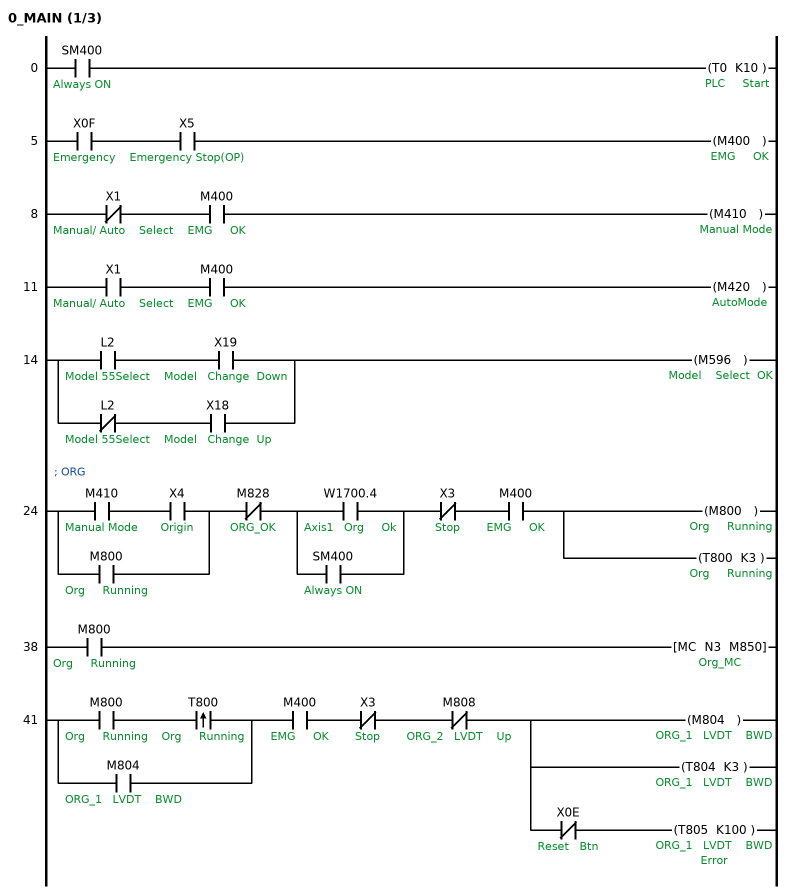
0     LD      SM400  ; Always ON
      OUT     T0 K10  ; PLC     Start
5     LD      X0F  ; Emergency
      AND     X5  ; Emergency Stop(OP)
      OUT     M400  ; EMG     OK
8     LDI     X1  ; Manual/ Auto    Select
      AND     M400  ; EMG     OK
      OUT     M410  ; Manual Mode
11    LD      X1  ; Manual/ Auto    Select
      AND     M400  ; EMG     OK
      OUT     M420  ; AutoMode
14    LD      L2  ; Model 55Select
      AND     X19  ; Model   Change  Down
      LDI     L2  ; Model 55Select
      AND     X18  ; Model   Change  Up
      ORB
      OUT     M596  ; Model    Select  OK
; ORG
24    LD      M410  ; Manual Mode
      AND     X4  ; Origin
      OR      M800  ; Org     Running
      ANI     M828  ; ORG_OK
      LD      W1700.4  ; Axis1   Org     Ok
      OR      SM400  ; Always ON
      ANB
      ANI     X3  ; Stop
      AND     M400  ; EMG     OK
      OUT     M800  ; Org     Running
      OUT     T800 K3  ; Org     Running
38    LD      M800  ; Org     Running
      MC      N3 M850  ; Org_MC
41    LD      M800  ; Org     Running
      ANDP    T800  ; Org     Running
      OR      M804  ; ORG_1   LVDT    BWD
      AND     M400  ; EMG     OK
      ANI     X3  ; Stop
      ANI     M808  ; ORG_2   LVDT    Up
      OUT     M804  ; ORG_1   LVDT    BWD
      OUT     T804 K3  ; ORG_1   LVDT    BWD
      ANI     X0E  ; Reset   Btn
      OUT     T805 K100  ; ORG_1   LVDT    BWD     Error
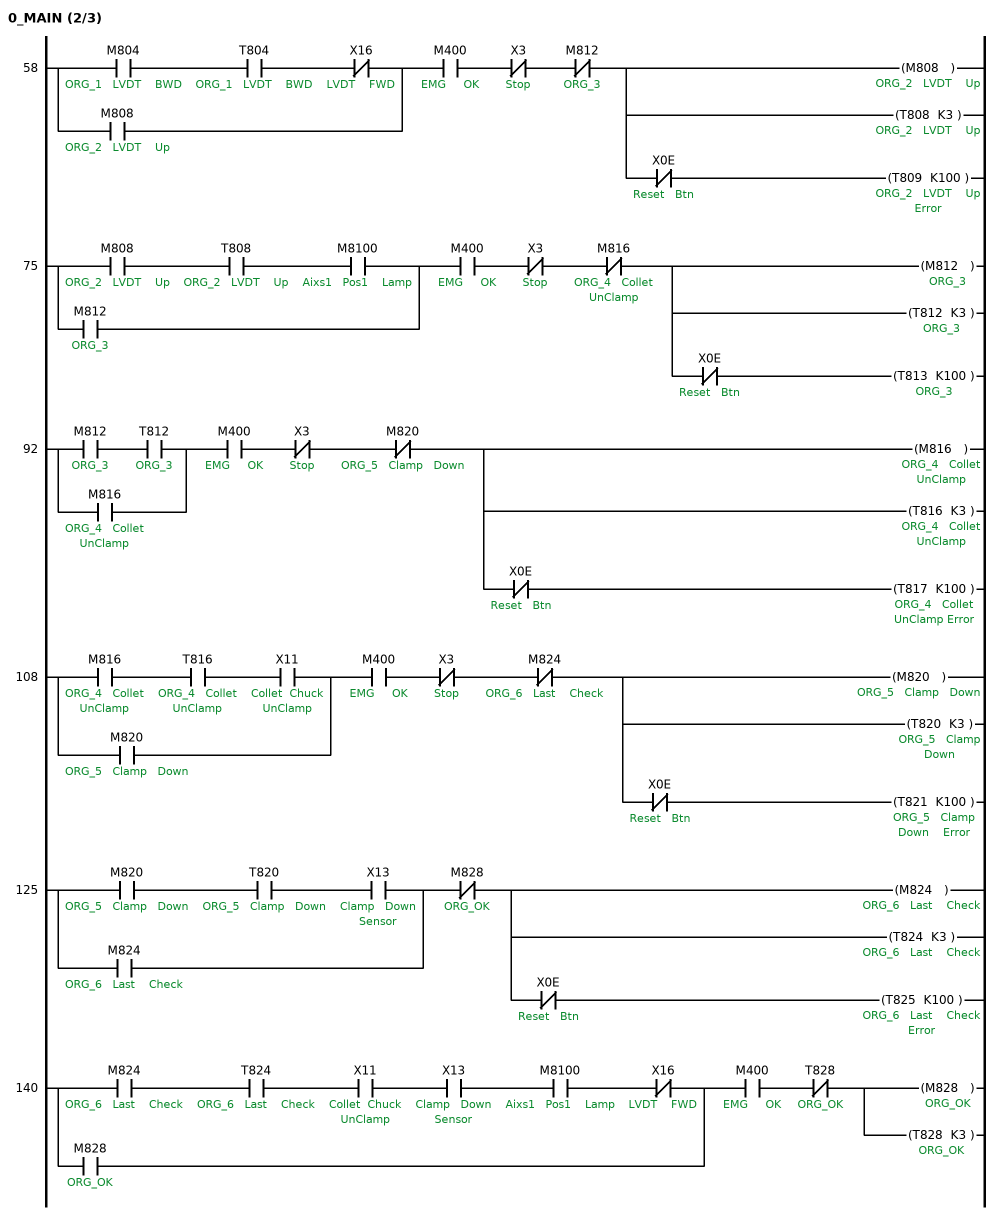
58    LD      M804  ; ORG_1   LVDT    BWD
      AND     T804  ; ORG_1   LVDT    BWD
      ANI     X16  ; LVDT    FWD
      OR      M808  ; ORG_2   LVDT    Up
      AND     M400  ; EMG     OK
      ANI     X3  ; Stop
      ANI     M812  ; ORG_3
      OUT     M808  ; ORG_2   LVDT    Up
      OUT     T808 K3  ; ORG_2   LVDT    Up
      ANI     X0E  ; Reset   Btn
      OUT     T809 K100  ; ORG_2   LVDT    Up      Error
75    LD      M808  ; ORG_2   LVDT    Up
      AND     T808  ; ORG_2   LVDT    Up
      AND     M8100  ; Aixs1   Pos1    Lamp
      OR      M812  ; ORG_3
      AND     M400  ; EMG     OK
      ANI     X3  ; Stop
      ANI     M816  ; ORG_4   Collet  UnClamp
      OUT     M812  ; ORG_3
      OUT     T812 K3  ; ORG_3
      ANI     X0E  ; Reset   Btn
      OUT     T813 K100  ; ORG_3
92    LD      M812  ; ORG_3
      AND     T812  ; ORG_3
      OR      M816  ; ORG_4   Collet  UnClamp
      AND     M400  ; EMG     OK
      ANI     X3  ; Stop
      ANI     M820  ; ORG_5   Clamp   Down
      OUT     M816  ; ORG_4   Collet  UnClamp
      OUT     T816 K3  ; ORG_4   Collet  UnClamp
      ANI     X0E  ; Reset   Btn
      OUT     T817 K100  ; ORG_4   Collet  UnClamp Error
108   LD      M816  ; ORG_4   Collet  UnClamp
      AND     T816  ; ORG_4   Collet  UnClamp
      AND     X11  ; Collet  Chuck   UnClamp
      OR      M820  ; ORG_5   Clamp   Down
      AND     M400  ; EMG     OK
      ANI     X3  ; Stop
      ANI     M824  ; ORG_6   Last    Check
      OUT     M820  ; ORG_5   Clamp   Down
      OUT     T820 K3  ; ORG_5   Clamp   Down
      ANI     X0E  ; Reset   Btn
      OUT     T821 K100  ; ORG_5   Clamp   Down    Error
125   LD      M820  ; ORG_5   Clamp   Down
      AND     T820  ; ORG_5   Clamp   Down
      AND     X13  ; Clamp   Down    Sensor
      OR      M824  ; ORG_6   Last    Check
      ANI     M828  ; ORG_OK
      OUT     M824  ; ORG_6   Last    Check
      OUT     T824 K3  ; ORG_6   Last    Check
      ANI     X0E  ; Reset   Btn
      OUT     T825 K100  ; ORG_6   Last    Check   Error
140   LD      M824  ; ORG_6   Last    Check
      AND     T824  ; ORG_6   Last    Check
      AND     X11  ; Collet  Chuck   UnClamp
      AND     X13  ; Clamp   Down    Sensor
      AND     M8100  ; Aixs1   Pos1    Lamp
      ANI     X16  ; LVDT    FWD
      OR      M828  ; ORG_OK
      AND     M400  ; EMG     OK
      ANI     T828  ; ORG_OK
      OUT     M828  ; ORG_OK
      OUT     T828 K3  ; ORG_OK
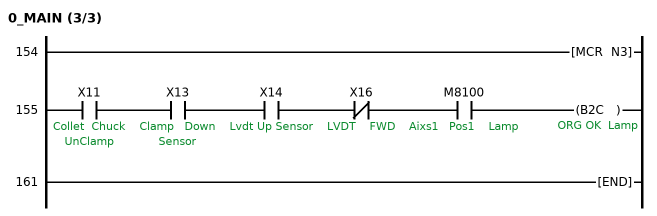
154   MCR     N3
155   LD      X11  ; Collet  Chuck   UnClamp
      AND     X13  ; Clamp   Down    Sensor
      AND     X14  ; Lvdt Up Sensor
      ANI     X16  ; LVDT    FWD
      AND     M8100  ; Aixs1   Pos1    Lamp
      OUT     B2C  ; ORG OK  Lamp
161   END
END_PROGRAM

PROGRAM 7_POSI
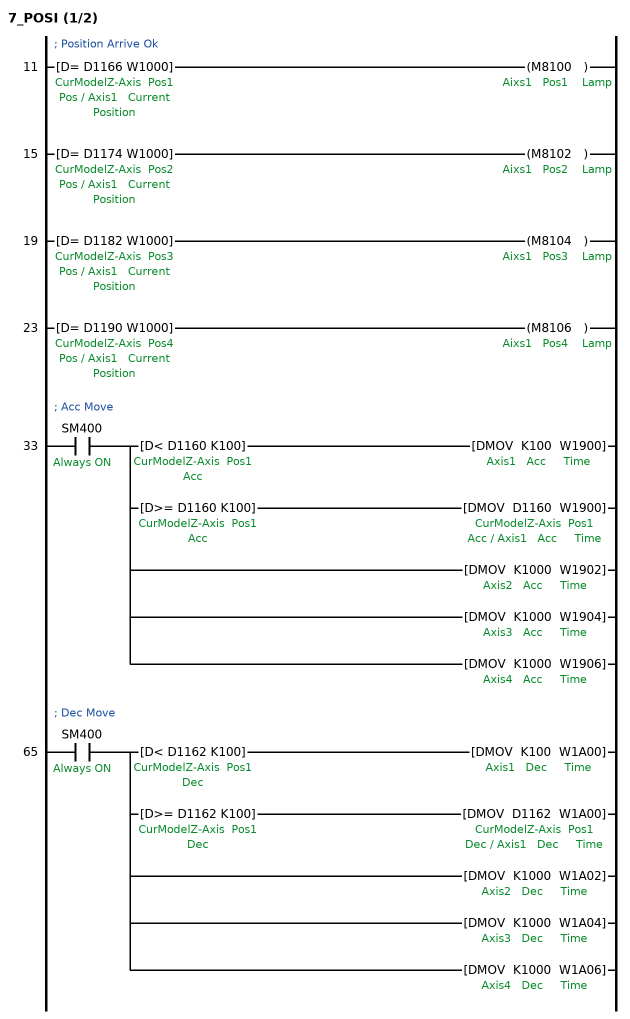
; Position Arrive Ok
11    LDD=    D1166 W1000  ; CurModelZ-Axis  Pos1    Pos / Axis1   Current Position
      OUT     M8100  ; Aixs1   Pos1    Lamp
15    LDD=    D1174 W1000  ; CurModelZ-Axis  Pos2    Pos / Axis1   Current Position
      OUT     M8102  ; Aixs1   Pos2    Lamp
19    LDD=    D1182 W1000  ; CurModelZ-Axis  Pos3    Pos / Axis1   Current Position
      OUT     M8104  ; Aixs1   Pos3    Lamp
23    LDD=    D1190 W1000  ; CurModelZ-Axis  Pos4    Pos / Axis1   Current Position
      OUT     M8106  ; Aixs1   Pos4    Lamp
; Acc Move
33    LD      SM400  ; Always ON
      MPS
      ANDD<   D1160 K100  ; CurModelZ-Axis  Pos1    Acc
      DMOV    K100 W1900  ; Axis1   Acc     Time
      MRD
      ANDD>=  D1160 K100  ; CurModelZ-Axis  Pos1    Acc
      DMOV    D1160 W1900
      MPP
      DMOV    K1000 W1902  ; Axis2   Acc     Time
      DMOV    K1000 W1904  ; Axis3   Acc     Time
      DMOV    K1000 W1906  ; Axis4   Acc     Time
; Dec Move
65    LD      SM400  ; Always ON
      MPS
      ANDD<   D1162 K100  ; CurModelZ-Axis  Pos1    Dec
      DMOV    K100 W1A00  ; Axis1   Dec     Time
      MRD
      ANDD>=  D1162 K100  ; CurModelZ-Axis  Pos1    Dec
      DMOV    D1162 W1A00
      MPP
      DMOV    K1000 W1A02  ; Axis2   Dec     Time
      DMOV    K1000 W1A04  ; Axis3   Dec     Time
      DMOV    K1000 W1A06  ; Axis4   Dec     Time
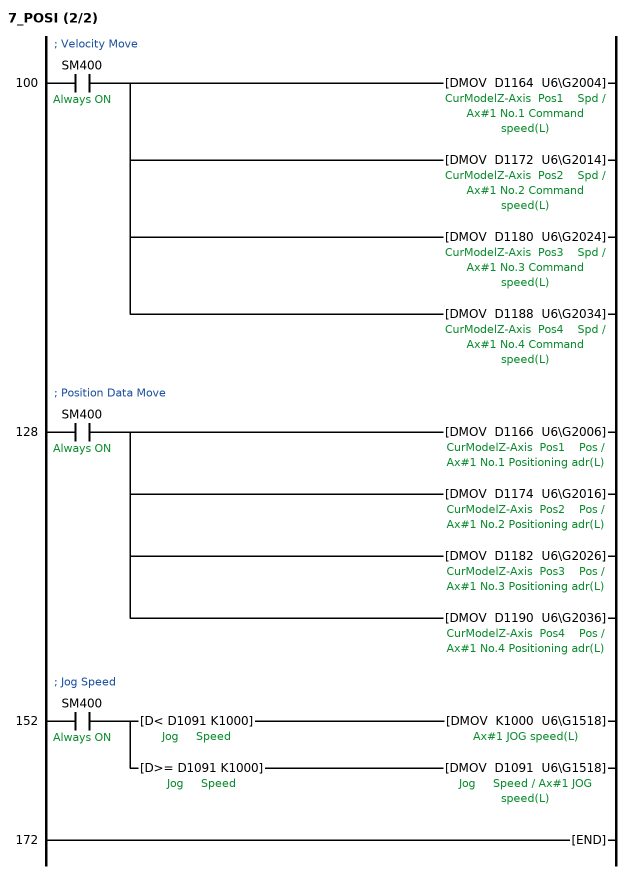
; Velocity Move
100   LD      SM400  ; Always ON
      DMOV    D1164 U6\G2004  ; CurModelZ-Axis  Pos1    Spd / Ax#1 No.1 Command speed(L)
      DMOV    D1172 U6\G2014  ; CurModelZ-Axis  Pos2    Spd / Ax#1 No.2 Command speed(L)
      DMOV    D1180 U6\G2024  ; CurModelZ-Axis  Pos3    Spd / Ax#1 No.3 Command speed(L)
      DMOV    D1188 U6\G2034  ; CurModelZ-Axis  Pos4    Spd / Ax#1 No.4 Command speed(L)
; Position Data Move
128   LD      SM400  ; Always ON
      DMOV    D1166 U6\G2006  ; Ax#1 No.1 Positioning adr(L)
      DMOV    D1174 U6\G2016  ; Ax#1 No.2 Positioning adr(L)
      DMOV    D1182 U6\G2026  ; Ax#1 No.3 Positioning adr(L)
      DMOV    D1190 U6\G2036  ; Ax#1 No.4 Positioning adr(L)
; Jog Speed
152   LD      SM400  ; Always ON
      MPS
      ANDD<   D1091 K1000  ; Jog     Speed
      DMOV    K1000 U6\G1518  ; Ax#1 JOG speed(L)
      MPP
      ANDD>=  D1091 K1000  ; Jog     Speed
      DMOV    D1091 U6\G1518
172   END
END_PROGRAM

PROGRAM 8_SERVO
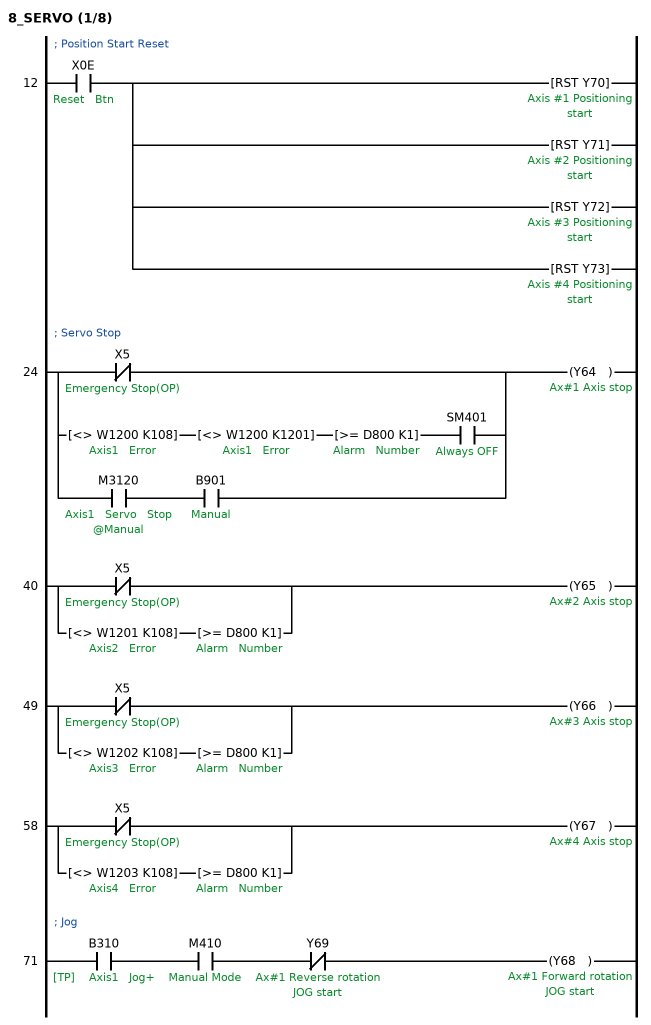
; Position Start Reset
12    LD      X0E  ; Reset   Btn
      RST     Y70  ; Axis #1 Positioning start
      RST     Y71  ; Axis #2 Positioning start
      RST     Y72  ; Axis #3 Positioning start
      RST     Y73  ; Axis #4 Positioning start
; Servo Stop
24    LDI     X5  ; Emergency Stop(OP)
      LD<>    W1200 K108  ; Axis1   Error
      AND<>   W1200 K1201  ; Axis1   Error
      AND>=   D800 K1  ; Alarm   Number
      AND     SM401  ; Always OFF
      ORB
      LD      M3120  ; Axis1   Servo   Stop    @Manual
      AND     B901  ; Manual
      ORB
      OUT     Y64  ; Ax#1 Axis stop
40    LDI     X5  ; Emergency Stop(OP)
      LD<>    W1201 K108  ; Axis2   Error
      AND>=   D800 K1  ; Alarm   Number
      ORB
      OUT     Y65  ; Ax#2 Axis stop
49    LDI     X5  ; Emergency Stop(OP)
      LD<>    W1202 K108  ; Axis3   Error
      AND>=   D800 K1  ; Alarm   Number
      ORB
      OUT     Y66  ; Ax#3 Axis stop
58    LDI     X5  ; Emergency Stop(OP)
      LD<>    W1203 K108  ; Axis4   Error
      AND>=   D800 K1  ; Alarm   Number
      ORB
      OUT     Y67  ; Ax#4 Axis stop
; Jog
71    LD      B310  ; [TP]    Axis1   Jog+
      AND     M410  ; Manual Mode
      ANI     Y69  ; Ax#1 Reverse rotation JOG start
      OUT     Y68  ; Ax#1 Forward rotation JOG start
